(* PLC project cb_ctd, Dassault Systèmes ControlBuild 2024x *)
(* stored: creationDateTime 2023-10-03T11:12:46-01:00 *)

(* This is a IEC 1131-3 counter. *)
FUNCTION_BLOCK timers_counters.cb_ctd
  VAR_INPUT
    CD : BOOL := false;
    LOAD : BOOL := false;
    PV : INT := 0;
  END_VAR
  VAR_OUTPUT
    QD : BOOL := false;
    CV : INT := 0;
  END_VAR


ACTION C_source_code:
/* -----------------------------------------------------------------	*/
/* Type : BFU									*/
/* Copyright : Geensoft							*/
/* Version : 1.0 23/03/2010							*/
/* -----------------------------------------------------------------	*/
/* This is a down-counter		(CTD)					*/
/* -------------------------------------------------------------	*/
if(LOAD) {
	CV = PV;
}
else {
	if(CD && (CV > -32768)) {
		CV = CV -1;
	}
}
QD = (CV <= 0);
END_ACTION
END_FUNCTION_BLOCK
